FUNCTION_BLOCK FB_SIMPLE
VAR_INPUT
	bPizzaDone : BOOL;
END_VAR
VAR_OUTPUT
	bLightOn : BOOL;
END_VAR
VAR
END_VAR

IF bPizzaDone THEN
	bLightOn := TRUE;
ELSE
	bLightOn := FALSE;
END_IF

END_FUNCTION_BLOCK

(* stored: Version 1.1.0.1, ProductVersion 3.1.4019.2
   POU FB_SIMPLE: Id {91874208-2b89-4cf9-b57b-9c2950ed7d8b}, SpecialFunc None *)
